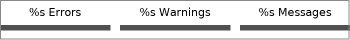
VISUALIZATION Uc_EventLogControl  // 350x40
    Rectangle (0,0 110x25), "%s Errors", text variable: stVisu.nErrorCount
        OnMouseClick: execute { stVisu.bFilterChanged := TRUE; stVisu.bErrorFilter := NOT stVisu.bErrorFilter; }
    Rectangle (0,25 110x5), colour toggle: stVisu.bErrorFilter, colour variable: stVisu.nErrorColor-16#c8000000
        p2167032090: stVisu.nErrorColor
    Rectangle (120,0 110x25), "%s Warnings", text variable: stVisu.nWarningCount
        OnMouseClick: execute { stVisu.bFilterChanged := TRUE; stVisu.bWarningFilter := NOT stVisu.bWarningFilter; }
    Rectangle (240,0 110x25), "%s Messages", text variable: stVisu.nInfoCount
        OnMouseClick: execute { stVisu.bFilterChanged := TRUE; stVisu.bInfoFilter := NOT stVisu.bInfoFilter; }
    Rectangle (120,25 110x5), colour toggle: stVisu.bWarningFilter, colour variable: stVisu.nWarningColor-16#c8000000
        p2167032090: stVisu.nWarningColor
    Rectangle (240,25 110x5), colour toggle: stVisu.bInfoFilter, colour variable: stVisu.nInfoColor-16#c8000000
        p2167032090: stVisu.nInfoColor
END_VISUALIZATION

(* stored: Version 1.1.0.1
   Visu Uc_EventLogControl: Id {954d78eb-e334-4007-a8a8-d13ce0311a4d} *)
